VAR_GLOBAL CONSTANT
    TcUnit_ResultExportXmlPath : T_MaxString :=
        'C:\TwinCAT\3.1\Boot\Plc\TcUnitResults.xml';
END_VAR

(* stored: Version 1.1.0.1
   GVL GVL_TcUnit: Id {5c05b202-c71e-4e7a-8375-cd62a7d43760} *)
